FUNCTION_BLOCK FB_SplitRealToWords_IEEE754
VAR_INPUT
	IN_Real : REAL;
END_VAR
VAR_OUTPUT
	OUT_WordStrong :  WORD;
	OUT_WordWeak :  WORD;

END_VAR
VAR

END_VAR

MEMCPY(destAddr := ADR(OUT_WordStrong), srcAddr := ADR(IN_Real), n := 2);
MEMCPY(destAddr := ADR(OUT_WordWeak), srcAddr := ADR(IN_Real) + 2, n := 2);

END_FUNCTION_BLOCK

(* stored: Version 1.1.0.1, ProductVersion 3.1.4024.6
   POU FB_SplitRealToWords_IEEE754: Id {049b6a07-c2f1-425d-b858-cf595a2af17e}, SpecialFunc None *)
